# EPICS autosave request: iocBoot/gmca_23b_ioc1/dbSave/fluoresCalib.req
$(P)$(MCA)_16384_gSl
$(P)$(MCA)_16384_itc
$(P)$(MCA)_16384_oSl

$(P)$(MCA)_8192_gSl
$(P)$(MCA)_8192_itc
$(P)$(MCA)_8192_oSl

$(P)$(MCA)_4096_gSl
$(P)$(MCA)_4096_itc
$(P)$(MCA)_4096_oSl

$(P)$(MCA)_2048_gSl
$(P)$(MCA)_2048_itc
$(P)$(MCA)_2048_oSl
